(* CODESYS project Untitled1_WithoutPlaceholder.library
   Company: MyCompany
   DefaultNamespace: MyDefaultNamespace
   Version: 6.7.8.9
   Placeholder: MyLibrary
   Author: MyAuthor
   Description: MyDescription
   Title: MyLibrary

Project tree, tasks and I/O mapping:
  libraries: Struckig, 0.9.3.0 (Stefan Besler); Tc2_Standard, * (Beckhoff Automation GmbH); Tc2_System, * (Beckhoff Automation GmbH); Tc3_Module, * (Beckhoff Automation GmbH); TcMatrix, 1.4.3 (Burks Engineering); TcTransform, 0.3.36 (Burks Engineering); TcLog, 0.3.1.0 (Benedikt Geisler); ZEquipment, 1.3.21.3 (Zeugwerk GmbH)
  DUTs/
  GVLs/
  POUs/
    program FB1 [ST]
    program MAIN [ST]
  VISUs/
*)

// POUs/FB1
PROGRAM FB1
VAR
  x : INT;
END_VAR

END_PROGRAM

// POUs/MAIN
PROGRAM MAIN
VAR
  x : INT := 5;
END_VAR

x := x + 1;

END_PROGRAM
